// TIA Portal V17 export
// export: Created 2023-05-07T12:12:12.0907637Z, ExportSetting WithDefaults, DisplayName Totally Integrated Automation Portal, DisplayVersion V17, DisplayName TIA Portal Openness, DisplayVersion V17, DisplayName TIA Portal Version Control Interface, DisplayVersion V17, DisplayName TIA Portal Test Suite Advanced, DisplayVersion V17, DisplayName STEP 7 Professional, DisplayVersion V17, DisplayName SIMATIC Energy Suite, DisplayVersion V17, DisplayName STEP 7 Safety, DisplayVersion V17, DisplayName WinCC Professional, DisplayVersion V17
FUNCTION "ConvertClass" : Void   // FC3, LAD
TITLE = ConvertClass
{ S7_Optimized_Access := 'TRUE' }
VERSION : 0.1
// stored: AutoNumber true, IsIECCheckEnabled false, SetENOAutomatically false, UDAEnableTagReadback false
   VAR_TEMP
      Output_PID_Real : Real;
      PV : Real;
      SP : Real;
      SPRamp : Real;
   END_VAR
BEGIN

REGION Network 1: Convert SetPoint: 0-300 -> 0-10
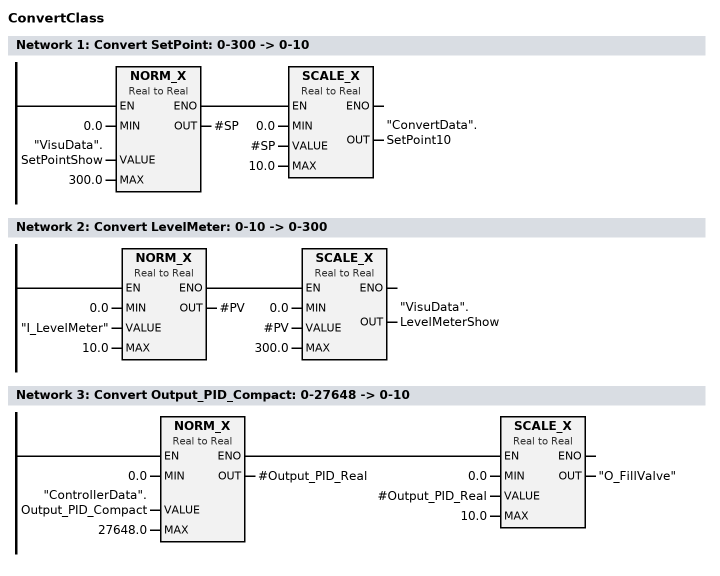
   RUNG wire#powerrail
      { S7_Templates := "[SrcType := Real, DestType := Real]" } Normalize(min := 0.0, value := "VisuData".SetPointShow, max := 300.0, out => #SP)
      { S7_Templates := "[SrcType := Real, DestType := Real]" } Scale(min := 0.0, value := #SP, max := 10.0, out => "ConvertData".SetPoint10)
   END_RUNG
   // the same network as SCL:
   #SP := NORM_X(MIN := 0.0, VALUE := "VisuData".SetPointShow, MAX := 300.0);
   "ConvertData".SetPoint10 := SCALE_X(MIN := 0.0, VALUE := #SP, MAX := 10.0);
END_REGION

REGION Network 2: Convert LevelMeter: 0-10 -> 0-300
   RUNG wire#powerrail
      { S7_Templates := "[SrcType := Real, DestType := Real]" } Normalize(min := 0.0, value := "I_LevelMeter", max := 10.0, out => #PV)
      { S7_Templates := "[SrcType := Real, DestType := Real]" } Scale(min := 0.0, value := #PV, max := 300.0, out => "VisuData".LevelMeterShow)
   END_RUNG
   // the same network as SCL:
   #PV := NORM_X(MIN := 0.0, VALUE := "I_LevelMeter", MAX := 10.0);
   "VisuData".LevelMeterShow := SCALE_X(MIN := 0.0, VALUE := #PV, MAX := 300.0);
END_REGION

REGION Network 3: Convert Output_PID_Compact: 0-27648 -> 0-10
   RUNG wire#powerrail
      { S7_Templates := "[SrcType := Real, DestType := Real]" } Normalize(min := 0.0, value := "ControllerData".Output_PID_Compact, max := 27648.0, out => #Output_PID_Real)
      { S7_Templates := "[SrcType := Real, DestType := Real]" } Scale(min := 0.0, value := #Output_PID_Real, max := 10.0, out => "O_FillValve")
   END_RUNG
   // the same network as SCL:
   #Output_PID_Real := NORM_X(MIN := 0.0, VALUE := "ControllerData".Output_PID_Compact, MAX := 27648.0);
   "O_FillValve" := SCALE_X(MIN := 0.0, VALUE := #Output_PID_Real, MAX := 10.0);
END_REGION
END_FUNCTION
